FUNCTION_BLOCK AOI_DI
VAR_INPUT
	ON: BOOL;
	OFF: BOOL;
	NAME: STRING := 'Not use';
	LINK: BOOL;
END_VAR
VAR_OUTPUT
	VALUE: BOOL;
	R_TRIG: BOOL;
	F_TRIG: BOOL;
END_VAR
VAR
	rtON: R_TRIG;
	rtOFF: R_TRIG;
	ftON: F_TRIG;
	ftOFF: F_TRIG;	
	rtValue: R_TRIG;
	ftValue: F_TRIG;

END_VAR

VALUE:= (ON OR LINK) AND NOT OFF; 
rtValue(CLK:=VALUE);
ftValue(CLK:=VALUE);
R_TRIG:=rtValue.Q;
F_TRIG:=ftValue.Q; 
rtON(CLK:=ON);
(*
IF rtON.Q THEN
	OFF:=FALSE;
	ON:=TRUE;	
END_IF
rtOFF(CLK:=OFF);
IF rtOFF.Q THEN
	ON:=FALSE;
	OFF:=TRUE;
END_IF

rtOFF(CLK:= OFF, Q=> );

IF ftOFF.Q THEN
	OFF:=FALSE;
END_IF

rtON(CLK:= ON, Q=> );

IF ftON.Q THEN
	ON:=FALSE;
END_IF

*)
IF ON AND OFF THEN
	ON:=FALSE;
	OFF:=FALSE;	
END_IF

END_FUNCTION_BLOCK

(* stored: Version 1.1.0.1, ProductVersion 3.1.4022.16
   POU AOI_DI: Id {6897fb74-1237-46d1-9bae-f3316086ec5e}, SpecialFunc None *)
